ABB RAPID module: RobotTargets.mod

MODULE RobotTargets
    CONST robtarget pHome:=[[935.00,0,1600],[0.00,0.0,-1,0],[-1,0,0,0],[0.400,9E+09,9E+09,9E+09,9E+09,9E+09]];
    !home position (Tool0 reference)

    CONST robtarget pHeli:=[[-1095.91,2234.75,149.91],[0.00275938,-0.707231,0.706972,-0.00259375],[1,-1,0,0],[0.41674,9E+09,9E+09,9E+09,9E+09,9E+09]];
    !Heli pickup
    CONST robtarget pVS:=[[261.28,2827.82,-79.82],[0.00814298,0.999961,0.000966756,0.00335392],[0,-1,-2,0],[0.415062,9E+09,9E+09,9E+09,9E+09,9E+09]];
    !VS pickup
    CONST robtarget pPlotter:=[[358.61,1298.35,-81.03],[0.00330879,0.66572,-0.746193,0.0013987],[0,0,-1,0],[-230.004,9E+09,9E+09,9E+09,9E+09,9E+09]];
    !Plotter pickup
    CONST robtarget pHTSHome:=[[-170.79,1515.79,1481.97],[0.00236128,0.676173,-0.736739,0.000524318],[0,0,0,0],[-230.006,9E+09,9E+09,9E+09,9E+09,9E+09]];
    CONST robtarget pVSTSHome:=[[-170.79,1515.79,1481.97],[0.00236128,0.676173,-0.736739,0.000524318],[0,0,0,0],[1200,9E+09,9E+09,9E+09,9E+09,9E+09]];
    CONST robtarget pHeliLid:=[[300,2000,1481.97],[0.00236128,0.676173,-0.736739,0.000524318],[0,0,0,0],[1200,9E+09,9E+09,9E+09,9E+09,9E+09]];
    CONST robtarget pVSLid:=[[-1100,1500,1500],[0.00814298,0.999961,0.000966756,0.00335392],[0,-1,-2,0],[-300,9E+09,9E+09,9E+09,9E+09,9E+09]];

    CONST robtarget ptHeli:=[[-1090.40,3326.52,-332.42],[0.000292045,-0.707231,0.706978,0.00234295],[1,-1,0,0],[0.419258,9E+09,9E+09,9E+09,9E+09,9E+09]];
    CONST robtarget ptHeliLid:=[[394.24,3085.52,994.74],[0.00461872,0.67616,-0.736727,-0.00450529],[1,0,0,0],[1200,9E+09,9E+09,9E+09,9E+09,9E+09]];

    PERS robtarget pTemp;

ENDMODULE
